INTERFACE IUnsupportedEventHandler EXTENDS IEventHandlerBase

END_INTERFACE

(* stored: Version 1.1.0.1, ProductVersion 3.1.4024.4
   Itf IUnsupportedEventHandler: Id {2c56818a-2ba9-466d-9719-ff833f58fa10} *)
